FUNCTION_BLOCK RingTokenMember (* Basic Function Block Type *)
  (* Standard: 61499-2 *)
  (* Version 0.2, 2003-12-04, JHC, Rockwell Automation, Renamed for better indexing. *)
  (* Version 0.1, 2002-11-05, JHC, Rockwell Automation, Corrected missing ST element in Algorithm REQ. *)
  (* Version 0.0, 2000-05-30, JHC, Rockwell Automation *)
  (* Compiler header: package fb.rt.cs725; *)
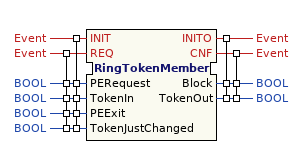
  EVENT_INPUT
    INIT WITH PERequest, TokenIn, PEExit, TokenJustChanged; (* Initialization Request *)
    REQ WITH PERequest, TokenIn, PEExit, TokenJustChanged; (* Normal Execution Request *)
  END_EVENT
  EVENT_OUTPUT
    INITO WITH Block, TokenOut; (* Initialization Confirm *)
    CNF WITH Block, TokenOut; (* Execution Confirmation *)
  END_EVENT
  VAR_INPUT
    PERequest : BOOL; (* Input event qualifier *)
    TokenIn : BOOL := false;
    PEExit : BOOL;
    TokenJustChanged : BOOL;
  END_VAR
  VAR_OUTPUT
    Block : BOOL; (* Output event qualifier *)
    TokenOut : BOOL;
  END_VAR
  VAR
    lastTokenIn : BOOL := true;
    lastPEExit : BOOL := 0;
    TokenChanged : BOOL := true;
  END_VAR
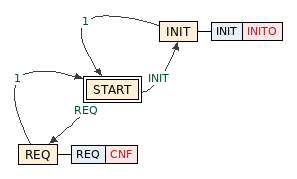
  EC_STATES
    START; (* Initial State *)
    INIT : INIT -> INITO; (* Initialization *)
    REQ : REQ -> CNF; (* Normal execution *)
  END_STATES
  EC_TRANSITIONS
    START TO INIT := INIT;
    INIT TO START := 1;
    START TO REQ := REQ;
    REQ TO START := 1;
  END_TRANSITIONS
  ALGORITHM INIT IN Java: (* Initialization algorithm *)
Block.value=false;
TokenOut.value=false;
System.out.println("init head, grant false, token true");
  END_ALGORITHM
  ALGORITHM REQ IN Java: (* Normally executed algorithm *)
System.out.println("3LastTokenIn, TokenIn, TokenOut:" + lastTokenIn.value + TokenIn.value + TokenOut.value);

if(TokenIn.value) {
if (TokenChanged.value) {
 if (!PERequest.value) {
  Block.value = false;
  TokenOut.value = false;
  System.out.println("Conv 3: I just got token, request is coming let bag go and keep token");
 } else {
  Block.value = false;
  TokenOut.value = true;
  System.out.println("Conv 3: I just got token, no request so run conveyer but let token go");
 }
} else {
 if (!PERequest.value) {
  System.out.println("Conv 3: I had token for a while, request here and bag passed eye, keep running conv and keep token");
  Block.value = false;
  TokenOut.value = false;
 } else {
  if (PEExit.value) {
   Block.value = false;
   TokenOut.value = true;
   System.out.println("Conv 3: I had token for a while, no requests and bag passed eye, let token go");
  } else {
   Block.value = false;
   TokenOut.value = false;
   System.out.println("Conv 3: I have token, no requests and bag not passed eye yet, keep token");
  }
 }
}
}

else {
    if (!PERequest.value) {
 Block.value = true;
TokenOut.value = true;
 System.out.println("Conv 3: No token, rquest here. Wait");
    }
else {
Block.value = false;
System.out.println("Conv 3: No token no request");
}
}

if(lastTokenIn.value != TokenIn.value) {
    TokenChanged.value = true;
}
else {
    TokenChanged.value = false;
}
lastTokenIn.value = TokenIn.value;
  END_ALGORITHM
END_FUNCTION_BLOCK
